{attribute 'linkalways'} 
{attribute 'no_explicit_call' := 'This FB is a CLASS and must be accessed using methods or properties'}
{attribute 'enable_dynamic_creation'}
FUNCTION_BLOCK FINAL ABS_WORD EXTENDS Node
VAR
	in : _WORD(0);
	out : _WORD(0);
END_VAR

METHOD PUBLIC Clone : I_Node
VAR
	pNode : POINTER TO ABS_WORD;
END_VAR
pNode := __NEW(ABS_WORD);
Clone := pNode^;
END_METHOD

METHOD FB_init : BOOL
VAR_INPUT
	bInitRetains : BOOL; // if TRUE, the retain variables are initialized (warm start / cold start)
	bInCopyCode : BOOL;  // if TRUE, the instance afterwards gets moved into the copy code (online change)
END_VAR
AddInput('in',THIS^.in);
AddOutput('out', THIS^.out);
END_METHOD

METHOD PROTECTED OnExecute
VAR
END_VAR
out.Value := ABS(in.Value);
END_METHOD

END_FUNCTION_BLOCK

(* stored: Version 1.1.0.1, ProductVersion 3.1.4024.15
   POU ABS_WORD: Id {566fbd70-5290-44e0-9f13-0f8e46b13ee6}, SpecialFunc None
   Folder Constructor: Id {31973259-56fd-417c-8bbc-d199737c1c6f}
   Method Clone: Id {49ba440d-a92b-4ac4-9a14-d523a526dfbb}
   Method FB_init: Id {7c1639a6-2a97-4f7b-94cf-d71e30f2f501}
   Method OnExecute: Id {f0f55d94-764c-48b8-81e0-61e4efc72ef3} *)
